METHOD PROTECTED sta_RUN : BOOL
VAR_INPUT
END_VAR
// state implemetation
//--------------------------------------------------------------------------------------
// Entry action
	IF (me.StateMachine.intState<>me.StateMachine.intStateLastCycle) THEN
		me.StateMachine.intStateLastCycle := me.StateMachine.intState;
	END_IF


//--------------------------------------------------------------------------------------
// Cyclic action
	IF (me.StateMachine.intState=me.StateMachine.intStateLastCycle) THEN
		// State Change Condition
		IF (NOT SIf.In.bolPumpOn.intern) AND (SIf.Cfg.VacuumPumpFeedback) THEN
			pfbAlarmCtrl^.setAlarm(CIf.Info.intCtrlId,INT_TO_UINT(E_ALM_VPC.VacuumPumpOnTimeout),0,ADR(SIf.Alm),E_AlmState.RST,CIf.Job.eMe_ActivAlmClass);
			me.StateMachine.intStateNext :=  BASE_PLC.cSTA_ERROR;
		END_IF;

		IF ((NOT SIf.In.bolVacuumOk.intern) AND (SIf.Cfg.VacuumSensorAvailable)) THEN
			pfbAlarmCtrl^.setAlarm(CIf.Info.intCtrlId,INT_TO_UINT(E_ALM_VPC.VacuumFailure),0,ADR(SIf.Alm),E_AlmState.RST,CIf.Job.eMe_ActivAlmClass);
			me.StateMachine.intStateNext :=  BASE_PLC.cSTA_ERROR;
		END_IF;	
	END_IF


//--------------------------------------------------------------------------------------
// Exit action
	IF (me.StateMachine.intState<>me.StateMachine.intStateNext) THEN
		;
	END_IF
END_METHOD

METHOD PROTECTED sta_RUNBusy : BOOL
VAR_INPUT
END_VAR
// state implemetation
//--------------------------------------------------------------------------------------
// Entry action
	IF (me.StateMachine.intState<>me.StateMachine.intStateLastCycle) THEN
		me.StateMachine.intStateLastCycle := me.StateMachine.intState;
		SIf.Out.bolVacuumPumpOn.intern := TRUE;

		fbSimulationTimer.IN := FALSE;
		fbSimulationTimer.PT := UDINT_TO_TIME(SIf.Par.udiSimVacuumPumpOnTime_ms);
		fbSimulationTimer(); // set time/reset timer
		fbSimulationTimer.IN := TRUE; // start timer
	END_IF


//--------------------------------------------------------------------------------------
// Cyclic action
	IF (me.StateMachine.intState=me.StateMachine.intStateLastCycle) THEN
		// Simulation
		IF (CIf.SwCfg.bolSimulation) THEN
			fbSimulationTimer(); // simulation time
			IF (fbSimulationTimer.Q) THEN
				SIf.In.bolPumpOn.intern := TRUE;
				SIf.In.bolVacuumOk.intern := TRUE;
			END_IF
		END_IF

		IF ((SIf.In.bolVacuumOk.intern) OR (NOT SIf.Cfg.VacuumPumpFeedback)) AND ((SIf.In.bolVacuumOk.intern) OR (NOT SIf.Cfg.VacuumSensorAvailable)) THEN
			me.StateMachine.intStateNext := VPC_CmdState.cSTA_VPC_StabilizeBusy;
		END_IF;		
		
		IF (me.StateMachine.udiTimeInState_ms > SIf.Par.udiVacuumPumpTime_ms) THEN
			IF (NOT SIf.In.bolPumpOn.intern) AND (SIf.Cfg.VacuumPumpFeedback) THEN
				pfbAlarmCtrl^.setAlarm(CIf.Info.intCtrlId,INT_TO_UINT(E_ALM_VPC.VacuumPumpOnTimeout),0,ADR(SIf.Alm),E_AlmState.RST,CIf.Job.eMe_ActivAlmClass);
			END_IF;

			IF ((NOT SIf.In.bolVacuumOk.intern) AND (SIf.Cfg.VacuumSensorAvailable)) THEN
				pfbAlarmCtrl^.setAlarm(CIf.Info.intCtrlId,INT_TO_UINT(E_ALM_VPC.VacuumFailure),0,ADR(SIf.Alm),E_AlmState.RST,CIf.Job.eMe_ActivAlmClass);
			END_IF;	

			me.StateMachine.intStateNext :=  cSTA_ERROR;
		END_IF
	END_IF


//--------------------------------------------------------------------------------------
// Exit action
	IF (me.StateMachine.intState<>me.StateMachine.intStateNext) THEN
		;
	END_IF
END_METHOD

METHOD PROTECTED sta_StabilizeVacuum : BOOL
VAR_INPUT
END_VAR
// state implemetation
//--------------------------------------------------------------------------------------
// Entry action
	IF (me.StateMachine.intState<>me.StateMachine.intStateLastCycle) THEN
		me.StateMachine.intStateLastCycle := me.StateMachine.intState;
	END_IF


//--------------------------------------------------------------------------------------
// Cyclic action
	IF (me.StateMachine.intState=me.StateMachine.intStateLastCycle) THEN
		// State Change Condition
		
		IF (me.StateMachine.udiTimeInState_ms > SIf.Par.udiVacuumStabilizationTime_ms) THEN
			me.StateMachine.intStateNext :=  BASE_PLC.cSTA_RUN;
		END_IF;	

		IF (NOT SIf.In.bolPumpOn.intern) AND (SIf.Cfg.VacuumPumpFeedback) THEN
			pfbAlarmCtrl^.setAlarm(CIf.Info.intCtrlId,INT_TO_UINT(E_ALM_VPC.VacuumPumpOnTimeout),0,ADR(SIf.Alm),E_AlmState.RST,CIf.Job.eMe_ActivAlmClass);
			me.StateMachine.intStateNext :=  BASE_PLC.cSTA_ERROR;
		END_IF;

		IF ((NOT SIf.In.bolVacuumOk.intern) AND (SIf.Cfg.VacuumSensorAvailable)) THEN
			pfbAlarmCtrl^.setAlarm(CIf.Info.intCtrlId,INT_TO_UINT(E_ALM_VPC.VacuumFailure),0,ADR(SIf.Alm),E_AlmState.RST,CIf.Job.eMe_ActivAlmClass);
			me.StateMachine.intStateNext :=  BASE_PLC.cSTA_ERROR;
		END_IF;	
	END_IF


//--------------------------------------------------------------------------------------
// Exit action
	IF (me.StateMachine.intState<>me.StateMachine.intStateNext) THEN
		;
	END_IF
END_METHOD

METHOD PROTECTED StateMachine : BOOL
SUPER^.StateMachine();

// main statemachine of base controller
CASE me.StateMachine.intState OF
    VPC_CmdState.cSTA_VPC_StabilizeBusy: 
        THIS^.sta_StabilizeVacuum();
	cSTA_RUNBusy: 
        THIS^.sta_RUNBusy();
    cSTA_RUN: 
        THIS^.sta_RUN();
END_CASE;
END_METHOD

END_FUNCTION_BLOCK
